// Mitsubishi GX Works2 project: 240402_인칭회로2   PLC: Q03UDV

PROGRAM MAIN
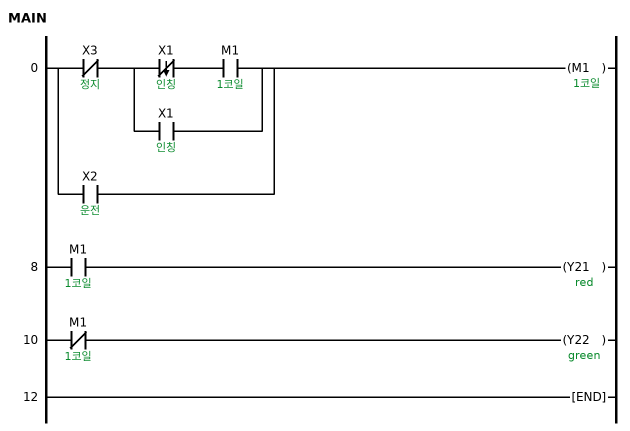
0     LDI     X3  ; 정지
      LDFI    X1  ; 인칭
      AND     M1  ; 1코일
      OR      X1  ; 인칭
      ANB
      OR      X2  ; 운전
      OUT     M1  ; 1코일
8     LD      M1  ; 1코일
      OUT     Y21  ; red
10    LDI     M1  ; 1코일
      OUT     Y22  ; green
12    END
END_PROGRAM
